PROGRAM MAIN
VAR
	conveyor : ConveyorSC_NC;
END_VAR

END_PROGRAM

(* stored: Version 1.1.0.1, ProductVersion 3.1.4024.11
   POU MAIN: Id {7f75ad39-54f6-4bc3-bace-5045f4922cc8}, SpecialFunc None *)
